// TIA Portal V17 export
// export: Created 2024-06-14T09:53:04.2858747Z, ExportSetting WithDefaults, DisplayName Totally Integrated Automation Portal, DisplayVersion V17, DisplayName TIA Portal Openness, DisplayVersion V17, DisplayName TIA Portal Version Control Interface, DisplayVersion V17, DisplayName Simotion SCOUT TIA, DisplayVersion 5.4.3.0, DisplayName SINAMICS Startdrive Advanced, DisplayVersion V17 SP1 Update 1, DisplayName SINAMICS Startdrive G110M, G120, G120C, G120D, G120P, G115D, DisplayVersion V17 SP1 Update 1, DisplayName SINAMICS Startdrive G130, G150, S120, S150, SINAMICS MV, S210, DisplayVersion V17 SP1 Update 1, DisplayName STEP 7 Professional, DisplayVersion V17, DisplayName STEP 7 Safety, DisplayVersion V17, DisplayName WinCC Professional, DisplayVersion V17
DATA_BLOCK "hmi_dummy_array"   // DB30
{ S7_Optimized_Access := 'TRUE' }
VERSION : 0.1
// stored: AutoNumber false, DBAccessibleFromOPCUA true, IsOnlyStoredInLoadMemory false, IsRetainMemResEnabled false, IsWriteProtectedInAS false, MemoryReserve 100
   VAR
      array_S1 { S7_SetPoint := 'True'} : Bool;
      array_S2 : Bool;
      S4_PrefillingDummyData { S7_SetPoint := 'True'} : Array[1..10] of "uCylinderData";
      LiftUpFeedback : Array[1..10] of Bool;
      DataransferDone : Bool;
      dummy : "uCylinderData";
      S5_PrefillingdummyData { S7_SetPoint := 'True'} : Array[1..10] of "uCylinderData";
      Gross_Weight { S7_SetPoint := 'True'} : Real;
      hmi_Desicion : Int;
      p_trig : Array[0..5] of Bool;
   END_VAR
BEGIN
   S4_PrefillingDummyData[1..3].iCylinderType := 0;
END_DATA_BLOCK
